{attribute 'qualified_only'}
VAR_GLOBAL CONSTANT
    // Arbitary cap on multidimensional states to simplify statements for the compiler.
    MAX_STATE_MOTORS: UINT := 3;
END_VAR

(* stored: Version 1.1.0.1
   GVL MotionConstants: Id {82935be4-17a5-42af-bb80-6817aae62409}, ParameterList True *)
